Universal Robots PolyScope program: asm_idler_pulley_p2.urp

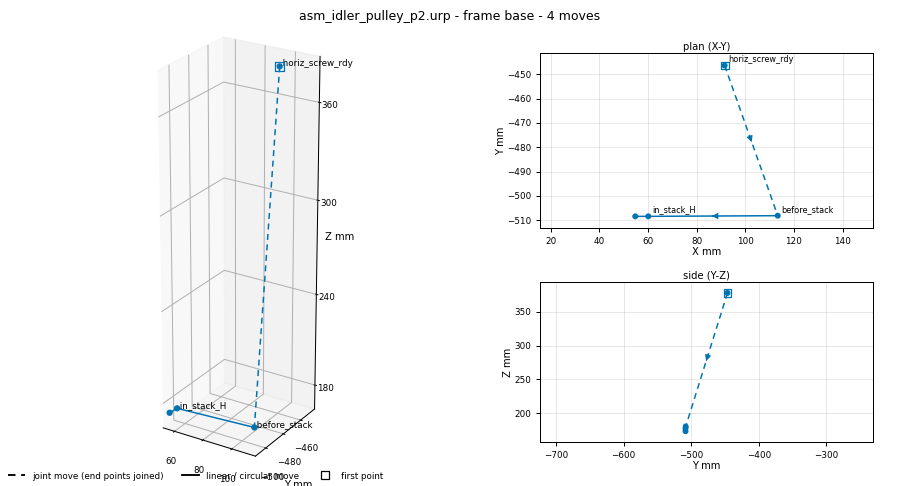
[picture p0: tool path of asm_idler_pulley_p2.urp in frame base, 4 of 4 moves have a stored position in this frame; points joined in program order, loops and branches not executed]
Program asm_idler_pulley_p2 (installation=default directory=/programs/wrs2020 createdIn=3.8.0.61336 lastSavedIn=5.10.0.106288 robotSerialNumber=20205500607)
Calibrated DH parameters: a=[0.000096, -0.337, -0.383372, 0.000118, 0.000015, 0]; d=[0.162724, 79.377998, -95.545185, 16.300583, 0.099689, 0.099499]; alpha=[1.569249, 0.003272, 0.005201, 1.570041, -1.570219, 0]; deltaTheta=[0, 0.65664, 5.410619, 0.215927, -0.000001, 0]
Robot Program (runOnlyOnce=true)
  MoveJ speed 60 deg/s, acceleration 80 deg/s^2 (useActiveTCP=true) feature=Base
    Waypoint horiz_screw_rdy: TCP in base x=91.509 y=-446.421 z=377.822 mm, rx=1.7333 ry=1.2228 rz=-1.2819 rad; joints [102.413, -107.496, 138.275, -189.231, -121.543, -259.619] deg; TCP offset x=0 y=0 z=165 mm, rx=0 ry=0 rz=0 rad
    Waypoint before_stack: TCP in base x=113.334 y=-508.169 z=180.394 mm, rx=2.1208 ry=1.7838 rz=-1.206 rad; joints [106.106, -83.335, 127.93, -164.755, -128.224, -254.548] deg
  MoveL speed 250 mm/s, acceleration 1200 mm/s^2 (useActiveTCP=true) feature=Base
    Waypoint in_stack_H: TCP in base x=60.113 y=-508.443 z=177.863 mm, rx=2.127 ry=1.7954 rz=-1.2032 rad; joints [98.708, -85.191, 131.571, -170.512, -124.339, -262.308] deg
  Popup Message (haltProgram=false message=wait for abot to open. c to incline slightly inputType=Text)
  MoveL speed 250 mm/s, acceleration 1200 mm/s^2 (useActiveTCP=true) feature=Base
    Waypoint Waypoint_10: TCP in base x=54.743 y=-508.443 z=173.386 mm, rx=2.122 ry=1.8043 rz=-1.2314 rad; joints [98.495, -84.166, 132.109, -172.492, -125.256, -263.374] deg
  Popup Message (haltProgram=false message=wait for washer and nut and fastening inputType=Text)
  Wait Sleep waitTime=1.5
